FUNCTION UpdateEventTimestampWithSystemTime
VAR_INPUT
	stEvent : ST_Event;
END_VAR
VAR_OUTPUT
	stEventOut : ST_Event;
END_VAR

(*Pass by value*)
stEventOut := stEvent;
stEventOut.dtTimestamp := // ...(GetSystemTime...)

END_FUNCTION

(* stored: Version 1.1.0.1, ProductVersion 3.1.4024.11
   POU UpdateEventTimestampWithSystemTime: Id {c72cb9da-759d-4038-87a1-8308f77b08cf}, SpecialFunc None *)
